(* PLC project Unnamed, Unknown Unnamed 1 *)
(* stored: creationDateTime 2022-08-16T15:49:17, modificationDateTime 2024-05-21T21:31:11 *)

PROGRAM Demo
  VAR
    DO1 AT %QX0.0 : BOOL;
    DO2 AT %QX0.1 : BOOL;
    DO3 AT %QX0.2 : BOOL;
    DO4 AT %QX0.3 : BOOL;
    DO5 AT %QX0.4 : BOOL;
    DO6 AT %QX0.5 : BOOL;
  END_VAR
  VAR
    TON0 : TON;
  END_VAR
  VAR
    DI1 AT %IX0.0 : BOOL;
    DI2 AT %IX0.1 : BOOL;
    DI3 AT %IX0.2 : BOOL;
    DI4 AT %IX0.3 : BOOL;
    DI5 AT %IX0.4 : BOOL;
    DI6 AT %IX0.5 : BOOL;
    DI7 AT %IX0.6 : BOOL;
    DI8 AT %IX0.7 : BOOL;
  END_VAR
  VAR
    RelayReset : BOOL;
    TON1 : TON;
    TON2 : TON;
    TON3 : TON;
    TON4 : TON;
    TON5 : TON;
  END_VAR

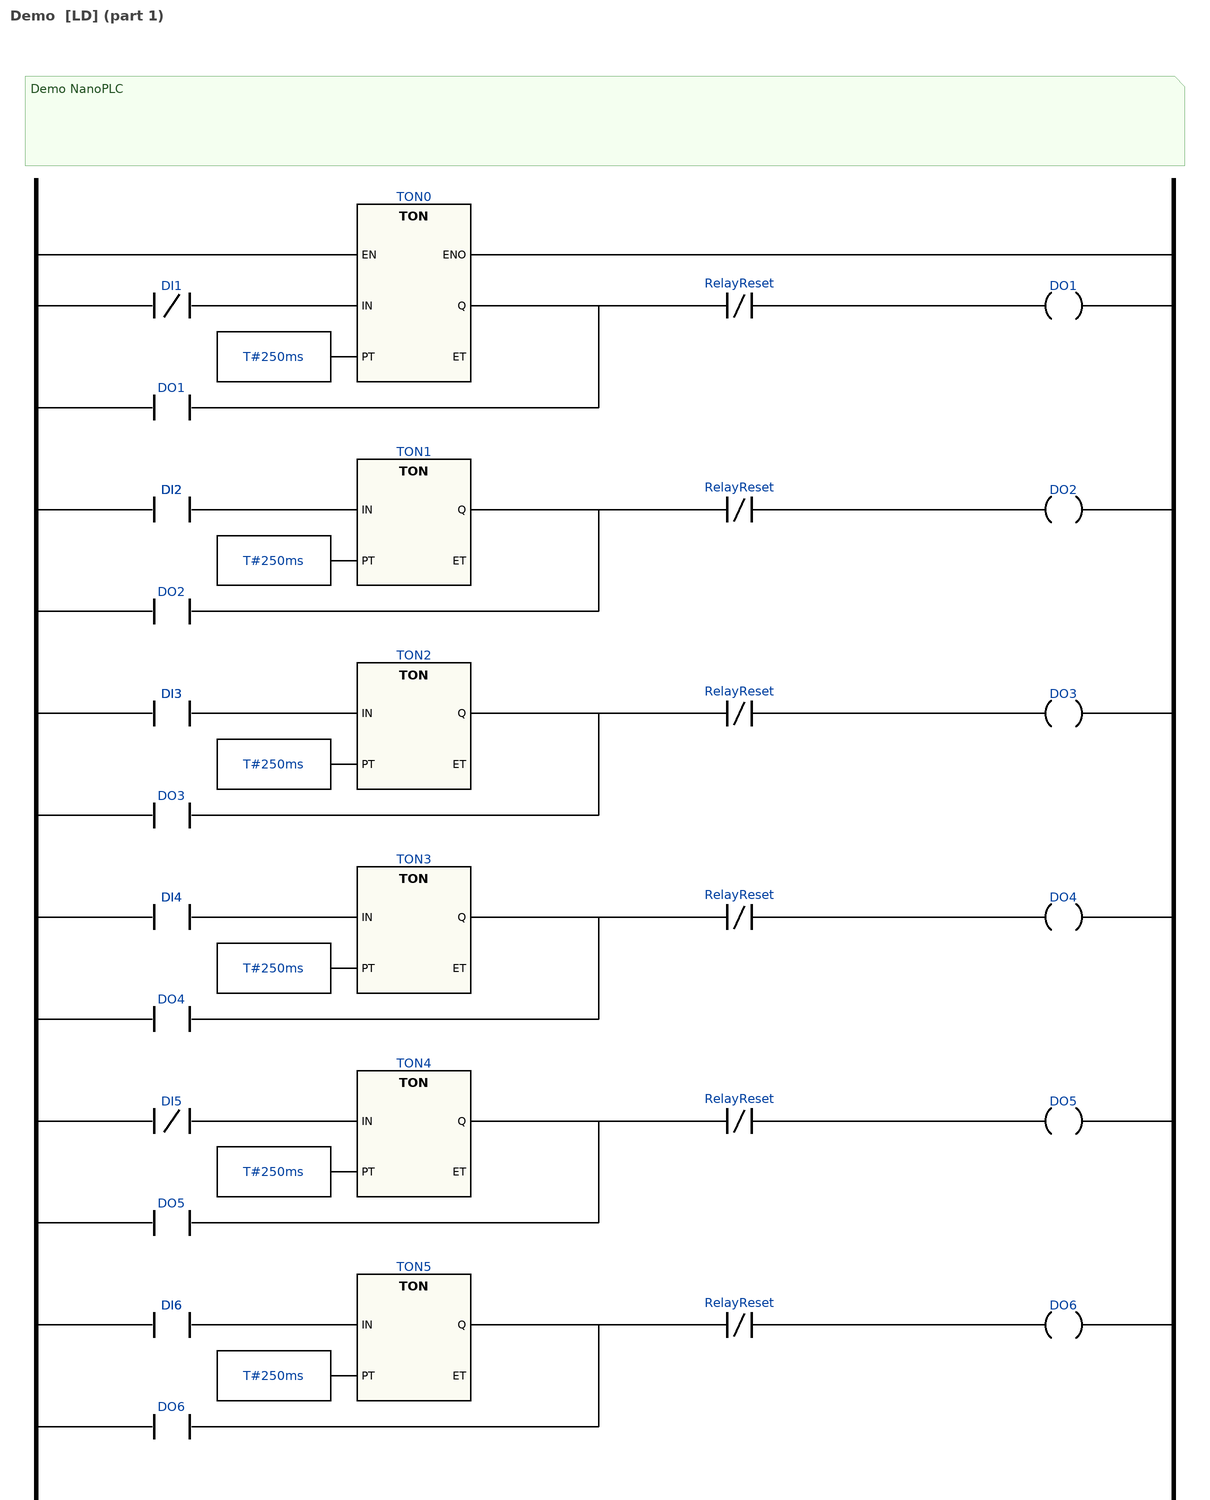
(* LD diagram, written out as Structured Text *)
(* Demo NanoPLC *)
TON0(IN := NOT DI1, PT := T#250ms);
DO1 := (TON0.Q OR DO1) AND NOT RelayReset;
TON1(IN := NOT DI2, PT := T#250ms);
DO2 := (TON1.Q OR DO2) AND NOT RelayReset;
TON2(IN := NOT DI3, PT := T#250ms);
DO3 := (TON2.Q OR DO3) AND NOT RelayReset;
TON3(IN := NOT DI4, PT := T#250ms);
DO4 := (TON3.Q OR DO4) AND NOT RelayReset;
TON4(IN := NOT DI5, PT := T#250ms);
DO5 := (TON4.Q OR DO5) AND NOT RelayReset;
TON5(IN := NOT DI6, PT := T#250ms);
DO6 := (TON5.Q OR DO6) AND NOT RelayReset;
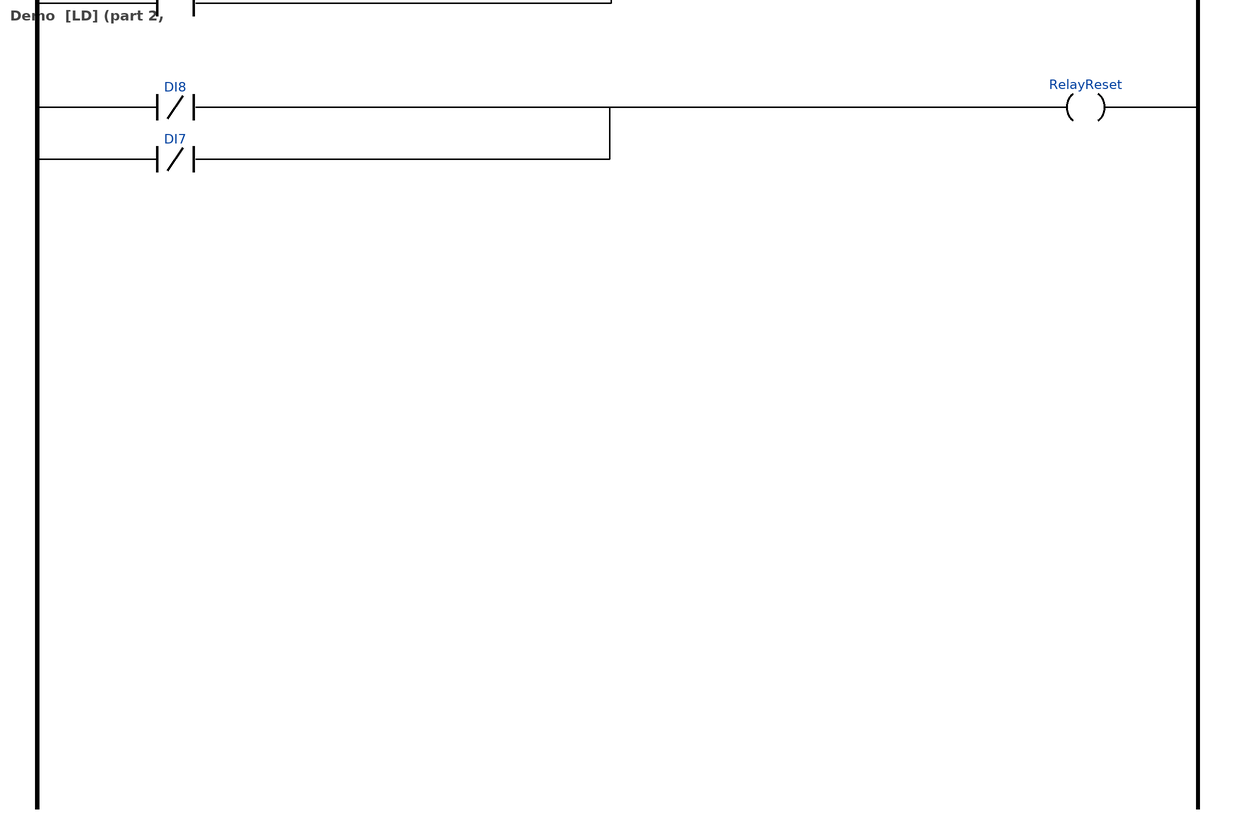
RelayReset := NOT DI7 OR NOT DI8;
(* drawn but not wired to any output: DI2, DI2, DI3, DI4, DI6 *)
END_PROGRAM

CONFIGURATION Config0
  RESOURCE Res0 ON PLC
    TASK task0(INTERVAL := T#20ms, PRIORITY := 0);
    PROGRAM instance0 WITH task0 : Demo;
  END_RESOURCE
END_CONFIGURATION
